// TwinCAT 3 PLC project Prog_Loops
// ProgramVersion: 3.1.4023.0
// libraries:
//   Tc2_Standard, * (Beckhoff Automation GmbH)
//   Tc2_System, * (Beckhoff Automation GmbH)
//   Tc3_Module, * (Beckhoff Automation GmbH)
// project tree:
//   / PlcTask.TcTTO
//   POUs/ MAIN.TcPOU, Prg_Loops.TcPOU
// real-time tasks:
//   TASK PlcTask: cycle T#10ms, priority 20, ADS port 350

CONFIGURATION Prog_Loops
    RESOURCE PLC ON TwinCAT3
        TASK PlcTask(INTERVAL := T#10ms, PRIORITY := 20);
        PROGRAM MAIN WITH PlcTask : MAIN;
    END_RESOURCE
END_CONFIGURATION

// ---- POUs/MAIN.TcPOU
PROGRAM MAIN
VAR
END_VAR

Prg_Loops();

END_PROGRAM

// ---- POUs/Prg_Loops.TcPOU
PROGRAM Prg_Loops
VAR
	Buttons: ARRAY[1..4] OF BOOL;
	AnalogSensor: ARRAY[1..4] OF INT := [5, 6, 7, 8];
	Coils: ARRAY[1..4] OF BOOL;
	
	i: INT;
END_VAR

FOR i:=1 TO 4 BY 1 DO
	IF Buttons[i] = TRUE AND AnalogSensor[i] > 6 THEN
		Coils[i]:=TRUE;
	ELSE
		Coils[i]:=FALSE;
	END_IF
END_FOR

END_PROGRAM
